{attribute 'GeneratedUsingTerminal: ELM3002-0000-0016'}
{attribute addProperty BoxType "ELM3002-0000-0016"}
{attribute addProperty Id "ARRAY_0DINT4"}
{attribute addProperty CRC "4065202250"}
{attribute addProperty Size "4"}
TYPE Samples_F24E104A :
STRUCT
	{attribute addProperty Name "ARRAY_0"}
	ARRAY_0 : DINT;
END_STRUCT
END_TYPE

(* stored: Version 1.2.0.0, ProductVersion 3.1.4024.9
   DUT Samples_F24E104A: Id {7ec130bc-cdc1-4393-92bd-ca7b44229670} *)
